// TIA Portal V19 export
FUNCTION_BLOCK "G120Comm"   // FB5, LAD
TITLE = Example of way to read and write the records in the G120
{ S7_Optimized_Access := 'TRUE' }
// stored: MemoryReserve 100, SetENOAutomatically false
   VAR_OUTPUT
      AnalogInput : Real;   // %
   END_VAR
   VAR
      WRREC_Instance { S7_SetPoint := 'True'} : WRREC;
      RDREC_Instance { S7_SetPoint := 'True'} : RDREC;
      WriteRecord : Struct
         Static_1 { S7_SetPoint := 'True'} : "HEADER";
         Static_2 { S7_SetPoint := 'True'} : "PARAMETERADDR";
      END_STRUCT;
      ReadRecord : Struct
         data : Array[0..5] of Byte;
         Value : Real;
      END_STRUCT;
   END_VAR
   // WriteRecord.Static_1.REQ_REF := 1;
   // WriteRecord.Static_1.REQ_ID := 1;
   // WriteRecord.Static_1.AXIS := 1;
   // WriteRecord.Static_1.NO_PARAM := 1;
   // WriteRecord.Static_2.ATTRIBUTE := 16;
   // WriteRecord.Static_2.NO_ELEM := 1;
   // WriteRecord.Static_2.PARA_NO := 755;
   // WriteRecord.Static_2.SUBINDEX := 0;
BEGIN
END_FUNCTION_BLOCK
